FUNCTION_BLOCK FB_DAC

VAR
	rAnaOut         :REAL;
	bFirstRun: BOOL := TRUE;
END_VAR
VAR_INPUT
	rDigitalIn			:			REAL	;		//数字量输入     例上位机
	rAnalogLowLMT		:			REAL	;		//模拟量下限     0
	rAanlogUpperLMT		:			REAL	;		//模拟量上限     32767
	rAnalogRef1			:			REAL	;		//参考点1：模拟量
	rDigitalRef1		:			REAL	;		//参考点1：数字量
	rAnalogRef2			:			REAL	;		//参考点2：模拟量
	rDigitalRef2		:			REAL	;		//参考点2：数字量
END_VAR
VAR_OUTPUT
	rAnalogOut			:			INT	    ;		//模拟量输出
	bError				:			BOOL	;		//错误
END_VAR

IF bFirstRun THEN
	IF ABS(rAnalogLowLMT) < 0.01 THEN
		rAanlogUpperLMT := -50000.0;
	END_IF;
	IF ABS(rAanlogUpperLMT) < 0.01 THEN
		rAanlogUpperLMT := 50000.0;
	END_IF;
END_IF;
bFirstRun:=FALSE;
IF rDigitalIn<>0 THEN
IF ABS(rAnalogRef2 - rAnalogRef1) > 0.00001 AND ABS(rDigitalRef2 - rDigitalRef1) >0.00001 THEN
	rAnaOut:=(rDigitalIn - rDigitalRef1) * (rAnalogRef2 - rAnalogRef1)/(rDigitalRef2 -rDigitalRef1) +rAnalogRef1;
	rAnaOut:=LIMIT(rAnalogLowLMT,rAnaOut,rAanlogUpperLMT);
	rAnalogOut:=REAL_TO_INT(rAnaOut);
	bError:=FALSE;
ELSE
	rAnalogOut := 0;
	bError     := TRUE;
END_IF;	
ELSE
rAnalogOut := 0;
END_IF;

END_FUNCTION_BLOCK

(* stored: Version 1.1.0.1, ProductVersion 3.1.4024.12
   POU FB_DAC: Id {03604c94-db96-415c-91fa-b99bc2d14561}, SpecialFunc None *)
